TYPE ST_Configuration :
STRUCT
	NUMBER_OF_JOINTS	: INT;
END_STRUCT
END_TYPE

(* stored: Version 1.1.0.1, ProductVersion 3.1.4024.9
   DUT ST_Configuration: Id {675c521e-6920-4694-8128-804f95be4939} *)
